(* CODESYS project CmpEmiconLog.library
   Author: Emicon
   Title: EmiconLog
   Version: 3.5.13.0
   Placeholder: PlaceholderTemplate
   DocFormat: reStructuredText
   Description: Emicon logging functionality
   Company: Emicon
   LanguageModelAttribute: qualified-access-only
   DefaultNamespace: EmLog

Project tree, tasks and I/O mapping:
  Libname/
    Enums/
      data type ERROR
    Function Blocks/
    Functions/
    GlobalConstants/
      global variables Constants
    GlobalVariables/
      global variables Variables
    Interfaces/
    Structs/
    Templates/
      function block ETrig [ST]
      function block ETrigA [ST]
      function block ETrigTl [ST]
      function block ETrigTlA [ST]
      function block ETrigTo [ST]
      function block ETrigToA [ST]
      function block ETrigToTl [ST]
      function block ETrigToTlA [ST]
      function block LTrig [ST]
    Types/
  function write_sys_log [ST]
  function write_ts_log [ST]
  function write_ti_log [ST]
  function clr_sys_log [ST]
  function create_log_files [ST]
  function get_next_log_item [ST]
*)

// Libname/Enums/ERROR
{attribute 'qualified_only'}
//{attribute 'conditionalshow' := 'SomeText'}
//{attribute 'conditionalshow'}
//{attribute 'hide'}
TYPE ERROR : (NO_ERROR, FIRST_ERROR, TIME_OUT, FIRST_MF, LAST_ERROR); END_TYPE

// Libname/GlobalConstants/Constants
{attribute 'qualified_only'}
//{attribute 'conditionalshow' := 'SomeText'}
//{attribute 'conditionalshow'}
//{attribute 'hide'}
VAR_GLOBAL CONSTANT
END_VAR

// Libname/GlobalVariables/Variables
{attribute 'qualified_only'}
//{attribute 'conditionalshow' := 'SomeText'}
//{attribute 'conditionalshow'}
//{attribute 'hide'}
VAR_GLOBAL
END_VAR

// Libname/Templates/ETrig
//{attribute 'hide_all_locals'}
//{attribute 'conditionalshow_all_locals' := 'SomeText'}
//{attribute 'conditionalshow_all_locals'}
//{attribute 'conditionalshow' := 'SomeText'}
//{attribute 'conditionalshow'}
//{attribute 'hide'}
FUNCTION_BLOCK ETrig
VAR_INPUT
	xExecute: BOOL;		(*	Rising edge: Action start
							Falling edge: Resets outputs
							If a falling edge occurs before the function block has completed its action, the outputs operate
							in the usual manner and are only reset if either the action is completed or
							in the event of an error. In this case, the corresponding output values (xDone, xError, iError)
							are present at the outputs for exactly one cycle.														*)
	(* specific Inputs *)
END_VAR
VAR_OUTPUT
	xDone: BOOL;		(*	Action successfully completed *)
	xBusy: BOOL;		(*	Function block active *)
	xError: BOOL;		(*	TRUE: error occurred, function block aborts action
							FALSE: no error	*)
	eError: ERROR;		(* If xError is true the eError is valid *)
	(* specific Outputs *)
END_VAR

END_FUNCTION_BLOCK

// Libname/Templates/ETrigA
//{attribute 'hide_all_locals'}
//{attribute 'conditionalshow_all_locals' := 'SomeText'}
//{attribute 'conditionalshow_all_locals'}
//{attribute 'conditionalshow' := 'SomeText'}
//{attribute 'conditionalshow'}
//{attribute 'hide'}
FUNCTION_BLOCK ETrigA
VAR_INPUT
	xExecute: BOOL;		(*	Rising edge: Action start
							Falling edge: Resets outputs
							If a falling edge occurs before the function block has completed its action, the outputs operate
							in the usual manner and are only reset if either the action is completed or aborted (xAbort), or
							in the event of an error. In this case, the corresponding output values (xDone, xError, iError)
							are present at the outputs for exactly one cycle. *)
	xAbort: BOOL;		(*	If this input is TRUE, the action is stopped immediately and all outputs are reset to their
							initial values.	*)
	(* specific Inputs *)
END_VAR
VAR_OUTPUT
	xDone: BOOL;		(*	Action successfully completed *)
	xBusy: BOOL;		(*	Function block active *)
	xError: BOOL;		(*	TRUE: error occurred, function block aborts action
							FALSE: no error	*)
	xAborted: BOOL;		(*	Action aborted by user*)
	eError: ERROR;		(* If xError is true the eError is valid *)
	(* specific Outputs *)
END_VAR

END_FUNCTION_BLOCK

// Libname/Templates/ETrigTl
//{attribute 'hide_all_locals'}
//{attribute 'conditionalshow_all_locals' := 'SomeText'}
//{attribute 'conditionalshow_all_locals'}
//{attribute 'conditionalshow' := 'SomeText'}
//{attribute 'conditionalshow'}
//{attribute 'hide'}
FUNCTION_BLOCK ETrigTl
VAR_INPUT
	xExecute: BOOL;		(*	Rising edge: Action start
							Falling edge: Resets outputs
							If a falling edge occurs before the function block has completed its action, the outputs operate
							in the usual manner and are only reset if either the action is completed or
							in the event of an error. In this case, the corresponding output values (xDone, xError, iError)
							are present at the outputs for exactly one cycle. *)
	udiTimeLimit: UDINT;	(*	This input defines how long (µs) an FB (requiring a long time for complete processing) may
								run until it is forced to return to the calling POU. The value 0 means that there is no
								time limitation. *)
	(* specific Inputs *)
END_VAR
VAR_OUTPUT
	xDone: BOOL;		(*	Action successfully completed *)
	xBusy: BOOL;		(*	Function block active *)
	xError: BOOL;		(*	TRUE: error occurred, function block aborts action
							FALSE: no error	*)
	eError: ERROR;		(* If xError is true the eError is valid *)
	(* specific Outputs *)
END_VAR

END_FUNCTION_BLOCK

// Libname/Templates/ETrigTlA
//{attribute 'hide_all_locals'}
//{attribute 'conditionalshow_all_locals' := 'SomeText'}
//{attribute 'conditionalshow_all_locals'}
//{attribute 'conditionalshow' := 'SomeText'}
//{attribute 'conditionalshow'}
//{attribute 'hide'}
FUNCTION_BLOCK ETrigTlA
VAR_INPUT
	xExecute: BOOL;		(*	Rising edge: Action start
							Falling edge: Resets outputs
							If a falling edge occurs before the function block has completed its action, the outputs operate
							in the usual manner and are only reset if either the action is completed or aborted (xAbort), or
							in the event of an error. In this case, the corresponding output values (xDone, xError, iError)
							are present at the outputs for exactly one cycle. *)
	xAbort: BOOL;			(*	If this input is TRUE, the action is stopped immediately and all outputs are reset to their
								initial values.	*)
	udiTimeLimit: UDINT;	(*	This input defines how long (µs) an FB (requiring a long time for complete processing) may
								run until it is forced to return to the calling POU. The value 0 means that there is no
								time limitation.																						*)
	(* specific Inputs *)
END_VAR
VAR_OUTPUT
	xDone: BOOL;		(*	Action successfully completed *)
	xBusy: BOOL;		(*	Function block active *)
	xError: BOOL;		(*	TRUE: error occurred, function block aborts action
							FALSE: no error	*)
	xAborted: BOOL;		(*	Action aborted by user*)
	eError: ERROR;		(* If xError is true the eError is valid *)
	(* specific Outputs *)
END_VAR

END_FUNCTION_BLOCK

// Libname/Templates/ETrigTo
//{attribute 'hide_all_locals'}
//{attribute 'conditionalshow_all_locals' := 'SomeText'}
//{attribute 'conditionalshow_all_locals'}
//{attribute 'conditionalshow' := 'SomeText'}
//{attribute 'conditionalshow'}
//{attribute 'hide'}
FUNCTION_BLOCK ETrigTo
VAR_INPUT
	xExecute: BOOL;		(*	Rising edge: Action start
							Falling edge: Resets outputs
							If a falling edge occurs before the function block has completed its action, the outputs operate
							in the usual manner and are only reset if either the action is completed or
							in the event of an error. In this case, the corresponding output values (xDone, xError, iError)
							are present at the outputs for exactly one cycle.														*)
	udiTimeOut: UDINT;	(*	This input defines the time (µs) after which an FB (e.g. requiring an external acknowledgement)
							aborts operation due to a timeout with error message. *)
	(* specific Inputs *)
END_VAR
VAR_OUTPUT
	xDone: BOOL;		(*	Action successfully completed *)
	xBusy: BOOL;		(*	Function block active *)
	xError: BOOL;		(*	TRUE: error occurred, function block aborts action
							FALSE: no error	*)
	eError: ERROR;		(* If xError is true the eError is valid *)
	(* specific Outputs *)
END_VAR

END_FUNCTION_BLOCK

// Libname/Templates/ETrigToA
//{attribute 'hide_all_locals'}
//{attribute 'conditionalshow_all_locals' := 'SomeText'}
//{attribute 'conditionalshow_all_locals'}
//{attribute 'conditionalshow' := 'SomeText'}
//{attribute 'conditionalshow'}
//{attribute 'hide'}
FUNCTION_BLOCK ETrigToA
VAR_INPUT
	xExecute: BOOL;		(*	Rising edge: Action start
								Falling edge: Resets outputs
								If a falling edge occurs before the function block has completed its action, the outputs operate
								in the usual manner and are only reset if either the action is completed or aborted (xAbort), or
								in the event of an error. In this case, the corresponding output values (xDone, xError, iError)
								are present at the outputs for exactly one cycle.														*)
	xAbort: BOOL;			(*	If this input is TRUE, the action is stopped immediately and all outputs are reset to their
								initial values.																							*)
	udiTimeOut: UDINT;	(*	This input defines the time (µs) after which an FB (e.g. requiring an external acknowledgement)
								aborts operation due to a timeout with error message.												*)
	(* specific Inputs *)
END_VAR
VAR_OUTPUT
	xDone: BOOL;		(*	Action successfully completed						*)
	xBusy: BOOL;		(*	Function block active									*)
	xError: BOOL;		(*	TRUE: error occurred, function block aborts action
							FALSE: no error										*)
	xAborted: BOOL;		(*	Action aborted by user*)
	eError: ERROR;		(* If xError is true the eError is valid *)
	(* specific Outputs *)
END_VAR

END_FUNCTION_BLOCK

// Libname/Templates/ETrigToTl
//{attribute 'hide_all_locals'}
//{attribute 'conditionalshow_all_locals' := 'SomeText'}
//{attribute 'conditionalshow_all_locals'}
//{attribute 'conditionalshow' := 'SomeText'}
//{attribute 'conditionalshow'}
//{attribute 'hide'}
FUNCTION_BLOCK ETrigToTl
VAR_INPUT
	xExecute: BOOL;		(*	Rising edge: Action start
							Falling edge: Resets outputs
							If a falling edge occurs before the function block has completed its action, the outputs operate
							in the usual manner and are only reset if either the action is completed or
							in the event of an error. In this case, the corresponding output values (xDone, xError, iError)
							are present at the outputs for exactly one cycle. *)
	udiTimeLimit: UDINT;	(*	This input defines how long (µs) an FB (requiring a long time for complete processing) may
								run until it is forced to return to the calling POU. The value 0 means that there is no
								time limitation. *)
	udiTimeOut: UDINT;	(*	This input defines the time (µs) after which an FB (e.g. requiring an external acknowledgement)
								aborts operation due to a timeout with error message. *)
	(* specific Inputs *)
END_VAR
VAR_OUTPUT
	xDone: BOOL;		(*	Action successfully completed *)
	xBusy: BOOL;		(*	Function block active *)
	xError: BOOL;		(*	TRUE: error occurred, function block aborts action
							FALSE: no error *)
	eError: ERROR;		(* If xError is true the eError is valid *)
	(* specific Outputs *)
END_VAR

END_FUNCTION_BLOCK

// Libname/Templates/ETrigToTlA
//{attribute 'hide_all_locals'}
//{attribute 'conditionalshow_all_locals' := 'SomeText'}
//{attribute 'conditionalshow_all_locals'}
//{attribute 'conditionalshow' := 'SomeText'}
//{attribute 'conditionalshow'}
//{attribute 'hide'}
FUNCTION_BLOCK ETrigToTlA
VAR_INPUT
	xExecute: BOOL;			(*	Rising edge: Action start
								Falling edge: Resets outputs
								If a falling edge occurs before the function block has completed its action, the outputs operate
								in the usual manner and are only reset if either the action is completed or aborted (xAbort), or
								in the event of an error. In this case, the corresponding output values (xDone, xError, iError)
								are present at the outputs for exactly one cycle. *)
	xAbort: BOOL;			(*	If this input is TRUE, the action is stopped immediately and all outputs are reset to their
								initial values.	*)
	udiTimeLimit: UDINT;	(*	This input defines how long (µs) an FB (requiring a long time for complete processing) may
								run until it is forced to return to the calling POU. The value 0 means that there is no
								time limitation.																						*)
	udiTimeOut: UDINT;		(*	This input defines the time (µs) after which an FB (e.g. requiring an external acknowledgement)
								aborts operation due to a timeout with error message.												*)
	(* specific Inputs *)
END_VAR
VAR_OUTPUT
	xDone: BOOL;		(*	Action successfully completed *)
	xBusy: BOOL;		(*	Function block active *)
	xError: BOOL;		(*	TRUE: error occurred, function block aborts action
							FALSE: no error	*)
	xAborted: BOOL;		(*	Action aborted by user*)
	eError: ERROR;		(* If xError is true the eError is valid *)
	(* specific Outputs *)
END_VAR

END_FUNCTION_BLOCK

// Libname/Templates/LTrig
//{attribute 'hide_all_locals'}
//{attribute 'conditionalshow_all_locals' := 'SomeText'}
//{attribute 'conditionalshow_all_locals'}
//{attribute 'conditionalshow' := 'SomeText'}
//{attribute 'conditionalshow'}
//{attribute 'hide'}
FUNCTION_BLOCK LTrig
VAR_INPUT
	xEnable: BOOL;	(*	TRUE: action running
						FALSE: action stopped, outputs xDone, xBusy, xError, iError are reset	*)
	(* specific Inputs *)
END_VAR
VAR_OUTPUT
	xDone: BOOL;		(*	Action successfully completed *)
	xBusy: BOOL;		(*	Function block active *)
	xError: BOOL;		(*	TRUE: error occurred, function block aborts action
							FALSE: no error	*)
	eError: ERROR;		(* If xError is true the eError is valid *)
	(* specific Outputs *)
END_VAR

END_FUNCTION_BLOCK

// write_sys_log
FUNCTION write_sys_log : UDINT
VAR_INPUT
	byClassId : BYTE;
	dwValue : DWORD;
END_VAR
VAR
END_VAR

END_FUNCTION

// write_ts_log
FUNCTION write_ts_log : UDINT
VAR_INPUT
	byClassId: BYTE;
	pbyData : POINTER TO BYTE;
END_VAR
VAR
END_VAR

END_FUNCTION

// write_ti_log
FUNCTION write_ti_log : UDINT
VAR_INPUT
	byClassId: BYTE;
	pbyData : POINTER TO BYTE;
END_VAR
VAR
END_VAR

END_FUNCTION

// clr_sys_log
FUNCTION clr_sys_log : UDINT
VAR_INPUT
END_VAR
VAR
END_VAR

END_FUNCTION

// create_log_files
FUNCTION create_log_files : DINT
VAR_INPUT
END_VAR
VAR
END_VAR

END_FUNCTION

// get_next_log_item
FUNCTION get_next_log_item : int
VAR_INPUT
	get_first : BOOL;
	log_str : POINTER TO STRING;
END_VAR
VAR
END_VAR

END_FUNCTION
